// TIA Portal V16 export
// export: Created 2021-11-12T13:31:14.9481279Z, ExportSetting WithDefaults, DisplayName Totally Integrated Automation Portal, DisplayVersion V16 Update 3, DisplayName TIA Portal Version Control Interface, DisplayVersion V16 Update 2, DisplayName TIA Portal Openness, DisplayVersion V16 Update 3, DisplayName SINAMICS Startdrive Advanced, DisplayVersion V16 Update 5, DisplayName SINAMICS Startdrive G130, G150, S120, S150, SINAMICS MV, S210, DisplayVersion V16 Update 5, DisplayName SINAMICS Startdrive G110M, G120, G120C, G120D, G120P, G115D, DisplayVersion V16 Update 5, DisplayName STEP 7 Professional, DisplayVersion V16 Update 3, DisplayName STEP 7 Safety, DisplayVersion V16, DisplayName WinCC UA Professional, DisplayVersion V16 Update 3
FUNCTION_BLOCK "STD_EuchnerDoor"   // FB77, LAD
{ S7_Optimized_Access := 'TRUE' }
VERSION : 0.1
// MICE STD Function Block
// STD_EuchnerDoor MGB2 module
// 
// Version                             Creation date                       Created by
// stored: AutoNumber true, IsIECCheckEnabled false, IsRetainMemResEnabled false, MemoryReserve 100, SetENOAutomatically false, UDAEnableTagReadback false
   VAR_INPUT
      IB_SubModule : "136687_UDT_MSM_Basic.Input";
      IB_LockModule : "UDT_MGB2-L/I_Extended.Input";
      IS_ZoneM : "UDT_Status_main";
      IS_ZoneS : "UDT_Zone_Status_specific";
      IB1LampTest : Bool;   // Lamp test button
      IB1Blinking_1Hz : Bool;   // Tact 1Hz
      IB1Blinking_2Hz : Bool;   // Tact 2Hz
      IB1AckReq : Bool;   // Alarms are resettable
      IB1UlckEn : Bool;   // Unlock enable
      IB1LckEn : Bool;   // Lock enable
      IB1LckMode : Bool;   // Lock mode - 1 can be lock before door is closed
      IB1Start : Bool;   // Start after zone was paused
      IB1AckRequestFromSafety : Bool;   // Safety block SFDoor needs ack
   END_VAR
   VAR_OUTPUT
      OS_Status : Struct
         Main : "UDT_Status_main";
         Specific : "UDT_Door_MGB2_L1_Status_specific";
         Error : "UDT_Error01";
      END_STRUCT;
      OB_SubModule : "136687_UDT_MSM.Output";
      OB_LockModule : "UDT_MGB-L/I.Output";
      OB1AckForSafety : Bool;   // Signal to Safety program
   END_VAR
   VAR
      SS_Alarm : Struct   // Device alarms
         SubModuleS1 : Bool;   // Sub module: Error S1
         LockModuleSM0 : Bool;   // Locking module: Error Sub module 0
         LockModuleSM1 : Bool;   // Locking module: Error Sub module 1
         LockModuleER : Bool;   // Locking module: Error escape release
         LockModuleG : Bool;   // Locking module: Error generally
         Res_0_5 : Bool;
         Res_0_6 : Bool;
         Res_0_7 : Bool;
         Res_1_0 : Bool;
         Res_1_1 : Bool;
         Res_1_2 : Bool;
         Res_1_3 : Bool;
         Res_1_4 : Bool;
         Res_1_5 : Bool;
         Res_1_6 : Bool;
         Res_1_7 : Bool;
      END_STRUCT;
      SS_Warning : Struct   // Device warnings
         Res_0_1 : Bool;
         Res_0_2 : Bool;
         Res_0_3 : Bool;
         Res_0_4 : Bool;
         Res_0_5 : Bool;
         Res_0_6 : Bool;
         Res_0_7 : Bool;
         Res_1_0 : Bool;
         Res_1_1 : Bool;
         Res_1_2 : Bool;
         Res_1_3 : Bool;
         Res_1_4 : Bool;
         Res_1_5 : Bool;
         Res_1_6 : Bool;
         Res_1_7 : Bool;
      END_STRUCT;
      SS_Edge : Array[0..9] of Bool;
      ST_PauseTON { S7_SetPoint := 'True'} : TON_TIME;   // Timer for pause
      ST_ACkSafetyTP : TP_TIME;   // Ack locked doors
      SB1CollError : Bool;   // Collective error from device
      SB1EStopLamp : Bool;   // E-Stop lamp
      SB0Lock : Bool;   // Lock signal (output)
      SB1RequestLock : Bool;   // Request to lock
      SB1RequestUnlock : Bool;   // Request to unlock
      SB1ResetLamp : Bool;   // Lock and reset alarm lamp
      SB1RequestLamp : Bool;   // Request to open lamp
      SB1RequestPause : Bool;   // Request to pause
      SB1ReadyToLock : Bool;
      SB1ReadyToOpen : Bool;
   END_VAR
   VAR_TEMP
      TS_Status : Struct
         Main : "UDT_Status_main";
         Specific : "UDT_Door_MGB2_L1_Status_specific";
         Error : "UDT_Error01";
      END_STRUCT;
   END_VAR
   VAR_TEMP   // added for the SCL form of the ladder/FBD networks
      _w1 : Bool;
   END_VAR
BEGIN

REGION Network 1: Clear temporary TS_Status - Main, Specific
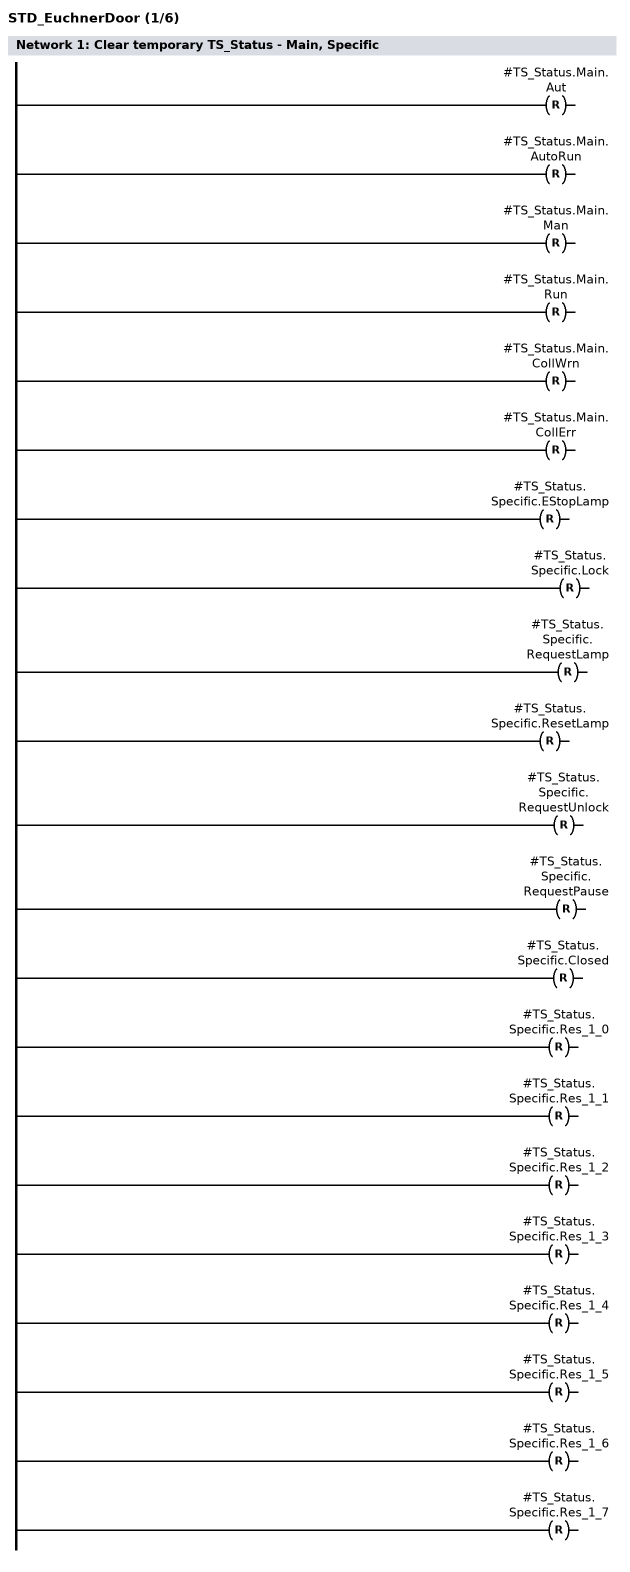
   RUNG wire#powerrail
      R_Coil( #TS_Status.Main.Aut )
   END_RUNG
   RUNG wire#powerrail
      R_Coil( #TS_Status.Main.AutoRun )
   END_RUNG
   RUNG wire#powerrail
      R_Coil( #TS_Status.Main.Man )
   END_RUNG
   RUNG wire#powerrail
      R_Coil( #TS_Status.Main.Run )
   END_RUNG
   RUNG wire#powerrail
      R_Coil( #TS_Status.Main.CollWrn )
   END_RUNG
   RUNG wire#powerrail
      R_Coil( #TS_Status.Main.CollErr )
   END_RUNG
   RUNG wire#powerrail
      R_Coil( #TS_Status.Specific.EStopLamp )
   END_RUNG
   RUNG wire#powerrail
      R_Coil( #TS_Status.Specific.Lock )
   END_RUNG
   RUNG wire#powerrail
      R_Coil( #TS_Status.Specific.RequestLamp )
   END_RUNG
   RUNG wire#powerrail
      R_Coil( #TS_Status.Specific.ResetLamp )
   END_RUNG
   RUNG wire#powerrail
      R_Coil( #TS_Status.Specific.RequestUnlock )
   END_RUNG
   RUNG wire#powerrail
      R_Coil( #TS_Status.Specific.RequestPause )
   END_RUNG
   RUNG wire#powerrail
      R_Coil( #TS_Status.Specific.Closed )
   END_RUNG
   RUNG wire#powerrail
      R_Coil( #TS_Status.Specific.Res_1_0 )
   END_RUNG
   RUNG wire#powerrail
      R_Coil( #TS_Status.Specific.Res_1_1 )
   END_RUNG
   RUNG wire#powerrail
      R_Coil( #TS_Status.Specific.Res_1_2 )
   END_RUNG
   RUNG wire#powerrail
      R_Coil( #TS_Status.Specific.Res_1_3 )
   END_RUNG
   RUNG wire#powerrail
      R_Coil( #TS_Status.Specific.Res_1_4 )
   END_RUNG
   RUNG wire#powerrail
      R_Coil( #TS_Status.Specific.Res_1_5 )
   END_RUNG
   RUNG wire#powerrail
      R_Coil( #TS_Status.Specific.Res_1_6 )
   END_RUNG
   RUNG wire#powerrail
      R_Coil( #TS_Status.Specific.Res_1_7 )
   END_RUNG
   // the same network as SCL:
   #TS_Status.Main.Aut := FALSE;
   #TS_Status.Main.AutoRun := FALSE;
   #TS_Status.Main.Man := FALSE;
   #TS_Status.Main.Run := FALSE;
   #TS_Status.Main.CollWrn := FALSE;
   #TS_Status.Main.CollErr := FALSE;
   #TS_Status.Specific.EStopLamp := FALSE;
   #TS_Status.Specific.Lock := FALSE;
   #TS_Status.Specific.RequestLamp := FALSE;
   #TS_Status.Specific.ResetLamp := FALSE;
   #TS_Status.Specific.RequestUnlock := FALSE;
   #TS_Status.Specific.RequestPause := FALSE;
   #TS_Status.Specific.Closed := FALSE;
   #TS_Status.Specific.Res_1_0 := FALSE;
   #TS_Status.Specific.Res_1_1 := FALSE;
   #TS_Status.Specific.Res_1_2 := FALSE;
   #TS_Status.Specific.Res_1_3 := FALSE;
   #TS_Status.Specific.Res_1_4 := FALSE;
   #TS_Status.Specific.Res_1_5 := FALSE;
   #TS_Status.Specific.Res_1_6 := FALSE;
   #TS_Status.Specific.Res_1_7 := FALSE;
END_REGION

REGION Network 2: Collective error of device
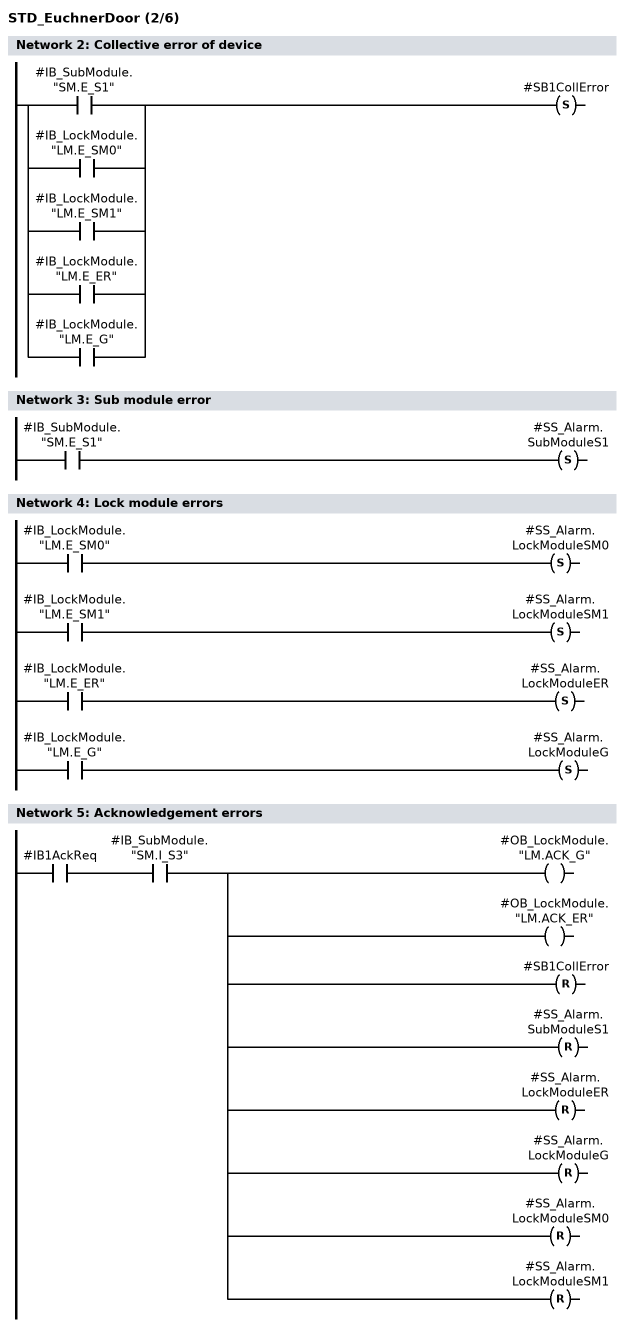
   RUNG wire#powerrail
      Contact( #IB_SubModule."SM.E_S1" )
      wire#w1
      S_Coil( #SB1CollError )
   END_RUNG
   RUNG wire#powerrail
      Contact( #IB_LockModule."LM.E_SM0" )
   END_RUNG wire#w1
   RUNG wire#powerrail
      Contact( #IB_LockModule."LM.E_SM1" )
   END_RUNG wire#w1
   RUNG wire#powerrail
      Contact( #IB_LockModule."LM.E_ER" )
   END_RUNG wire#w1
   RUNG wire#powerrail
      Contact( #IB_LockModule."LM.E_G" )
   END_RUNG wire#w1
   // the same network as SCL:
   IF #IB_SubModule."SM.E_S1" OR #IB_LockModule."LM.E_SM0" OR #IB_LockModule."LM.E_SM1" OR #IB_LockModule."LM.E_ER" OR #IB_LockModule."LM.E_G" THEN
       #SB1CollError := TRUE;
   END_IF;
END_REGION

REGION Network 3: Sub module error
   RUNG wire#powerrail
      Contact( #IB_SubModule."SM.E_S1" )
      S_Coil( #SS_Alarm.SubModuleS1 )
   END_RUNG
   // the same network as SCL:
   IF #IB_SubModule."SM.E_S1" THEN #SS_Alarm.SubModuleS1 := TRUE; END_IF;
END_REGION

REGION Network 4: Lock module errors
   RUNG wire#powerrail
      Contact( #IB_LockModule."LM.E_SM0" )
      S_Coil( #SS_Alarm.LockModuleSM0 )
   END_RUNG
   RUNG wire#powerrail
      Contact( #IB_LockModule."LM.E_SM1" )
      S_Coil( #SS_Alarm.LockModuleSM1 )
   END_RUNG
   RUNG wire#powerrail
      Contact( #IB_LockModule."LM.E_ER" )
      S_Coil( #SS_Alarm.LockModuleER )
   END_RUNG
   RUNG wire#powerrail
      Contact( #IB_LockModule."LM.E_G" )
      S_Coil( #SS_Alarm.LockModuleG )
   END_RUNG
   // the same network as SCL:
   IF #IB_LockModule."LM.E_SM0" THEN #SS_Alarm.LockModuleSM0 := TRUE; END_IF;
   IF #IB_LockModule."LM.E_SM1" THEN #SS_Alarm.LockModuleSM1 := TRUE; END_IF;
   IF #IB_LockModule."LM.E_ER" THEN #SS_Alarm.LockModuleER := TRUE; END_IF;
   IF #IB_LockModule."LM.E_G" THEN #SS_Alarm.LockModuleG := TRUE; END_IF;
END_REGION

REGION Network 5: Acknowledgement errors
   RUNG wire#powerrail
      Contact( #IB1AckReq )
      Contact( #IB_SubModule."SM.I_S3" )
      wire#w1
      Coil( #OB_LockModule."LM.ACK_G" )
   END_RUNG
   RUNG wire#w1
      Coil( #OB_LockModule."LM.ACK_ER" )
   END_RUNG
   RUNG wire#w1
      R_Coil( #SB1CollError )
   END_RUNG
   RUNG wire#w1
      R_Coil( #SS_Alarm.SubModuleS1 )
   END_RUNG
   RUNG wire#w1
      R_Coil( #SS_Alarm.LockModuleER )
   END_RUNG
   RUNG wire#w1
      R_Coil( #SS_Alarm.LockModuleG )
   END_RUNG
   RUNG wire#w1
      R_Coil( #SS_Alarm.LockModuleSM0 )
   END_RUNG
   RUNG wire#w1
      R_Coil( #SS_Alarm.LockModuleSM1 )
   END_RUNG
   // the same network as SCL:
   #OB_LockModule."LM.ACK_G" := #IB1AckReq AND #IB_SubModule."SM.I_S3";
   #OB_LockModule."LM.ACK_ER" := #OB_LockModule."LM.ACK_G";
   IF #OB_LockModule."LM.ACK_G" THEN
       #SB1CollError := FALSE;
       #SS_Alarm.SubModuleS1 := FALSE;
       #SS_Alarm.LockModuleER := FALSE;
       #SS_Alarm.LockModuleG := FALSE;
       #SS_Alarm.LockModuleSM0 := FALSE;
       #SS_Alarm.LockModuleSM1 := FALSE;
   END_IF;
END_REGION

REGION Network 6: Red lamp - E-Stop
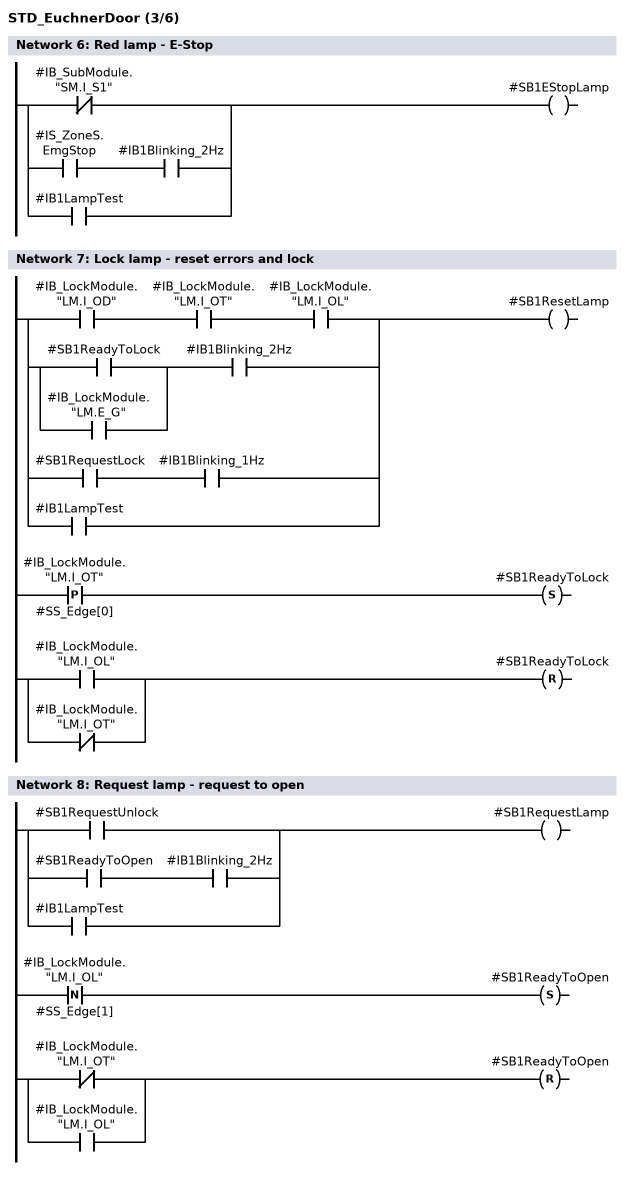
   RUNG wire#powerrail
      I_Contact( #IB_SubModule."SM.I_S1" )
      wire#w1
      Coil( #SB1EStopLamp )
   END_RUNG
   RUNG wire#powerrail
      Contact( #IS_ZoneS.EmgStop )
      Contact( #IB1Blinking_2Hz )
   END_RUNG wire#w1
   RUNG wire#powerrail
      Contact( #IB1LampTest )
   END_RUNG wire#w1
   // the same network as SCL:
   #SB1EStopLamp := NOT #IB_SubModule."SM.I_S1" OR (#IS_ZoneS.EmgStop AND #IB1Blinking_2Hz) OR #IB1LampTest;
END_REGION

REGION Network 7: Lock lamp - reset errors and lock
   RUNG wire#powerrail
      Contact( #IB_LockModule."LM.I_OD" )
      Contact( #IB_LockModule."LM.I_OT" )
      Contact( #IB_LockModule."LM.I_OL" )
      wire#w1
      Coil( #SB1ResetLamp )
   END_RUNG
   RUNG wire#powerrail
      Contact( #SB1ReadyToLock )
      wire#w2
      Contact( #IB1Blinking_2Hz )
   END_RUNG wire#w1
   RUNG wire#powerrail
      Contact( #IB_LockModule."LM.E_G" )
   END_RUNG wire#w2
   RUNG wire#powerrail
      Contact( #SB1RequestLock )
      Contact( #IB1Blinking_1Hz )
   END_RUNG wire#w1
   RUNG wire#powerrail
      Contact( #IB1LampTest )
   END_RUNG wire#w1
   RUNG wire#powerrail
      P_Contact(operand := #IB_LockModule."LM.I_OT", bit := #SS_Edge[0])
      S_Coil( #SB1ReadyToLock )
   END_RUNG
   RUNG wire#powerrail
      Contact( #IB_LockModule."LM.I_OL" )
      wire#w3
      R_Coil( #SB1ReadyToLock )
   END_RUNG
   RUNG wire#powerrail
      I_Contact( #IB_LockModule."LM.I_OT" )
   END_RUNG wire#w3
   // the same network as SCL:
   #SB1ResetLamp := (#IB_LockModule."LM.I_OD" AND #IB_LockModule."LM.I_OT" AND #IB_LockModule."LM.I_OL") OR ((#SB1ReadyToLock OR #IB_LockModule."LM.E_G") AND #IB1Blinking_2Hz) OR (#SB1RequestLock AND #IB1Blinking_1Hz) OR #IB1LampTest;
   #_w1 := #IB_LockModule."LM.I_OT" AND NOT #SS_Edge[0];   // rising edge of #IB_LockModule."LM.I_OT"
   #SS_Edge[0] := #IB_LockModule."LM.I_OT";
   IF #_w1 THEN #SB1ReadyToLock := TRUE; END_IF;
   IF #IB_LockModule."LM.I_OL" OR NOT #IB_LockModule."LM.I_OT" THEN #SB1ReadyToLock := FALSE; END_IF;
END_REGION

REGION Network 8: Request lamp - request to open
   RUNG wire#powerrail
      Contact( #SB1RequestUnlock )
      wire#w1
      Coil( #SB1RequestLamp )
   END_RUNG
   RUNG wire#powerrail
      Contact( #SB1ReadyToOpen )
      Contact( #IB1Blinking_2Hz )
   END_RUNG wire#w1
   RUNG wire#powerrail
      Contact( #IB1LampTest )
   END_RUNG wire#w1
   RUNG wire#powerrail
      N_Contact(operand := #IB_LockModule."LM.I_OL", bit := #SS_Edge[1])
      S_Coil( #SB1ReadyToOpen )
   END_RUNG
   RUNG wire#powerrail
      I_Contact( #IB_LockModule."LM.I_OT" )
      wire#w2
      R_Coil( #SB1ReadyToOpen )
   END_RUNG
   RUNG wire#powerrail
      Contact( #IB_LockModule."LM.I_OL" )
   END_RUNG wire#w2
   // the same network as SCL:
   #SB1RequestLamp := #SB1RequestUnlock OR (#SB1ReadyToOpen AND #IB1Blinking_2Hz) OR #IB1LampTest;
   #_w1 := NOT #IB_LockModule."LM.I_OL" AND #SS_Edge[1];   // falling edge of #IB_LockModule."LM.I_OL"
   #SS_Edge[1] := #IB_LockModule."LM.I_OL";
   IF #_w1 THEN #SB1ReadyToOpen := TRUE; END_IF;
   IF NOT #IB_LockModule."LM.I_OT" OR #IB_LockModule."LM.I_OL" THEN #SB1ReadyToOpen := FALSE; END_IF;
END_REGION

REGION Network 9: Request to lock
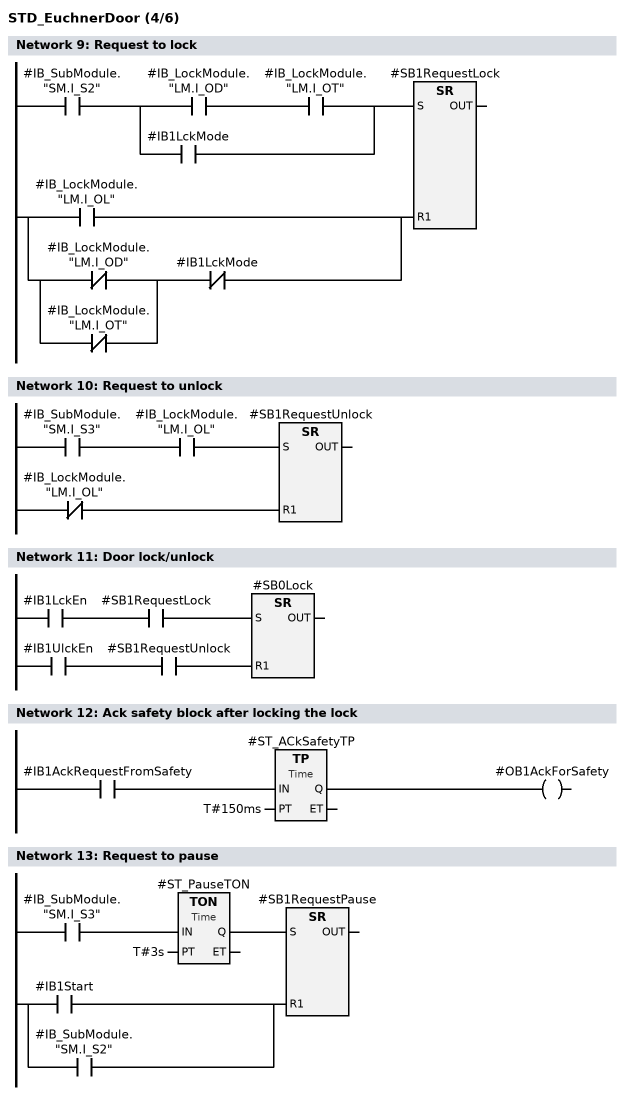
   RUNG wire#powerrail
      Contact( #IB_SubModule."SM.I_S2" )
      wire#w1
      Contact( #IB_LockModule."LM.I_OD" )
      Contact( #IB_LockModule."LM.I_OT" )
      wire#w2
      S_SR(operand := #SB1RequestLock, r1 := wire#w4)
   END_RUNG
   RUNG wire#w1
      Contact( #IB1LckMode )
   END_RUNG wire#w2
   RUNG wire#powerrail
      Contact( #IB_LockModule."LM.I_OL" )
   END_RUNG wire#w4
   RUNG wire#powerrail
      I_Contact( #IB_LockModule."LM.I_OD" )
      wire#w3
      I_Contact( #IB1LckMode )
   END_RUNG wire#w4
   RUNG wire#powerrail
      I_Contact( #IB_LockModule."LM.I_OT" )
   END_RUNG wire#w3
   // the same network as SCL:
   IF #IB_SubModule."SM.I_S2" AND ((#IB_LockModule."LM.I_OD" AND #IB_LockModule."LM.I_OT") OR #IB1LckMode) THEN
       #SB1RequestLock := TRUE;   // SR flip-flop
   END_IF;
   IF #IB_LockModule."LM.I_OL" OR ((NOT #IB_LockModule."LM.I_OD" OR NOT #IB_LockModule."LM.I_OT") AND NOT #IB1LckMode) THEN
       #SB1RequestLock := FALSE;
   END_IF;
END_REGION

REGION Network 10: Request to unlock
   RUNG wire#powerrail
      Contact( #IB_SubModule."SM.I_S3" )
      Contact( #IB_LockModule."LM.I_OL" )
      S_SR(operand := #SB1RequestUnlock, r1 := wire#w1)
   END_RUNG
   RUNG wire#powerrail
      I_Contact( #IB_LockModule."LM.I_OL" )
   END_RUNG wire#w1
   // the same network as SCL:
   IF #IB_SubModule."SM.I_S3" AND #IB_LockModule."LM.I_OL" THEN
       #SB1RequestUnlock := TRUE;   // SR flip-flop
   END_IF;
   IF NOT #IB_LockModule."LM.I_OL" THEN #SB1RequestUnlock := FALSE; END_IF;
END_REGION

REGION Network 11: Door lock/unlock
   RUNG wire#powerrail
      Contact( #IB1LckEn )
      Contact( #SB1RequestLock )
      S_SR(operand := #SB0Lock, r1 := wire#w1)
   END_RUNG
   RUNG wire#powerrail
      Contact( #IB1UlckEn )
      Contact( #SB1RequestUnlock )
   END_RUNG wire#w1
   // the same network as SCL:
   IF #IB1LckEn AND #SB1RequestLock THEN
       #SB0Lock := TRUE;   // SR flip-flop
   END_IF;
   IF #IB1UlckEn AND #SB1RequestUnlock THEN #SB0Lock := FALSE; END_IF;
END_REGION

REGION Network 12: Ack safety block after locking the lock
   RUNG wire#powerrail
      Contact( #IB1AckRequestFromSafety )
      { S7_Templates := "time_type := Time" } #ST_ACkSafetyTP.TP(pt := T#150ms, et =>)
      Coil( #OB1AckForSafety )
   END_RUNG
   // the same network as SCL:
   #ST_ACkSafetyTP(IN := #IB1AckRequestFromSafety, PT := T#150ms);   // TP
   #OB1AckForSafety := #ST_ACkSafetyTP.Q;
END_REGION

REGION Network 13: Request to pause
   RUNG wire#powerrail
      Contact( #IB_SubModule."SM.I_S3" )
      { S7_Templates := "time_type := Time" } #ST_PauseTON.TON(pt := T#3s, et =>)
      S_SR(operand := #SB1RequestPause, r1 := wire#w1)
   END_RUNG
   RUNG wire#powerrail
      Contact( #IB1Start )
   END_RUNG wire#w1
   RUNG wire#powerrail
      Contact( #IB_SubModule."SM.I_S2" )
   END_RUNG wire#w1
   // the same network as SCL:
   #ST_PauseTON(IN := #IB_SubModule."SM.I_S3", PT := T#3s);   // TON
   IF #ST_PauseTON.Q THEN
       #SB1RequestPause := TRUE;   // SR flip-flop
   END_IF;
   IF #IB1Start OR #IB_SubModule."SM.I_S2" THEN #SB1RequestPause := FALSE; END_IF;
END_REGION

REGION Network 14: Copy static variables to output variables
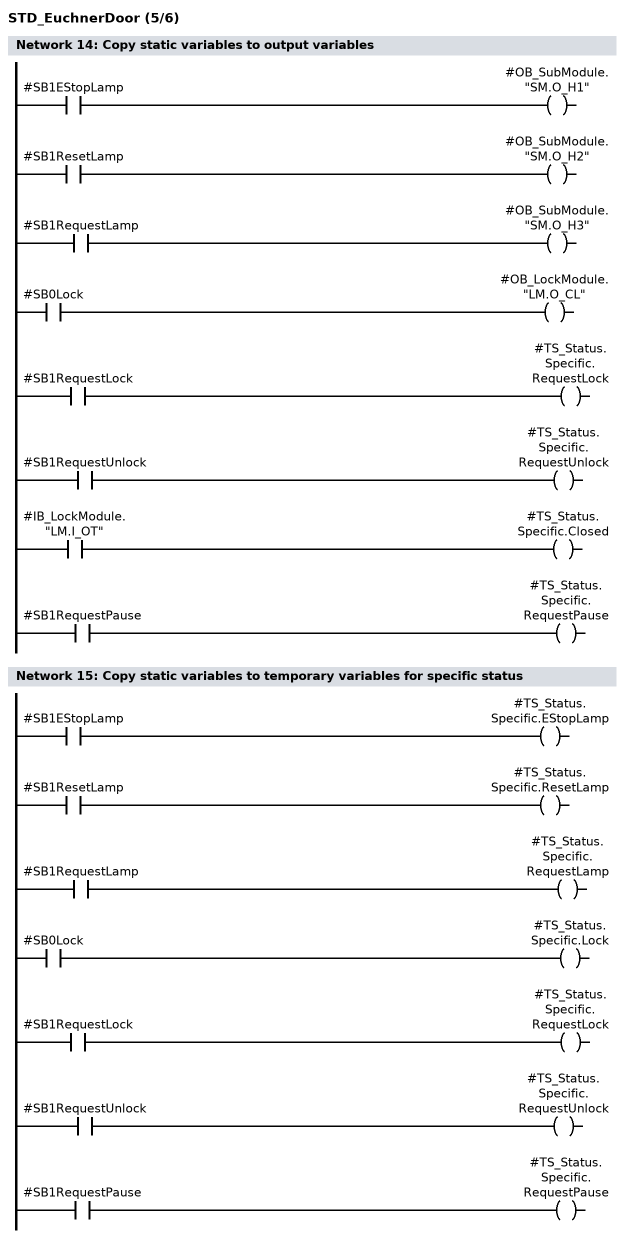
   RUNG wire#powerrail
      Contact( #SB1EStopLamp )
      Coil( #OB_SubModule."SM.O_H1" )
   END_RUNG
   RUNG wire#powerrail
      Contact( #SB1ResetLamp )
      Coil( #OB_SubModule."SM.O_H2" )
   END_RUNG
   RUNG wire#powerrail
      Contact( #SB1RequestLamp )
      Coil( #OB_SubModule."SM.O_H3" )
   END_RUNG
   RUNG wire#powerrail
      Contact( #SB0Lock )
      Coil( #OB_LockModule."LM.O_CL" )
   END_RUNG
   RUNG wire#powerrail
      Contact( #SB1RequestLock )
      Coil( #TS_Status.Specific.RequestLock )
   END_RUNG
   RUNG wire#powerrail
      Contact( #SB1RequestUnlock )
      Coil( #TS_Status.Specific.RequestUnlock )
   END_RUNG
   RUNG wire#powerrail
      Contact( #IB_LockModule."LM.I_OT" )
      Coil( #TS_Status.Specific.Closed )
   END_RUNG
   RUNG wire#powerrail
      Contact( #SB1RequestPause )
      Coil( #TS_Status.Specific.RequestPause )
   END_RUNG
   // the same network as SCL:
   #OB_SubModule."SM.O_H1" := #SB1EStopLamp;
   #OB_SubModule."SM.O_H2" := #SB1ResetLamp;
   #OB_SubModule."SM.O_H3" := #SB1RequestLamp;
   #OB_LockModule."LM.O_CL" := #SB0Lock;
   #TS_Status.Specific.RequestLock := #SB1RequestLock;
   #TS_Status.Specific.RequestUnlock := #SB1RequestUnlock;
   #TS_Status.Specific.Closed := #IB_LockModule."LM.I_OT";
   #TS_Status.Specific.RequestPause := #SB1RequestPause;
END_REGION

REGION Network 15: Copy static variables to temporary variables for specific status
   RUNG wire#powerrail
      Contact( #SB1EStopLamp )
      Coil( #TS_Status.Specific.EStopLamp )
   END_RUNG
   RUNG wire#powerrail
      Contact( #SB1ResetLamp )
      Coil( #TS_Status.Specific.ResetLamp )
   END_RUNG
   RUNG wire#powerrail
      Contact( #SB1RequestLamp )
      Coil( #TS_Status.Specific.RequestLamp )
   END_RUNG
   RUNG wire#powerrail
      Contact( #SB0Lock )
      Coil( #TS_Status.Specific.Lock )
   END_RUNG
   RUNG wire#powerrail
      Contact( #SB1RequestLock )
      Coil( #TS_Status.Specific.RequestLock )
   END_RUNG
   RUNG wire#powerrail
      Contact( #SB1RequestUnlock )
      Coil( #TS_Status.Specific.RequestUnlock )
   END_RUNG
   RUNG wire#powerrail
      Contact( #SB1RequestPause )
      Coil( #TS_Status.Specific.RequestPause )
   END_RUNG
   // the same network as SCL:
   #TS_Status.Specific.EStopLamp := #SB1EStopLamp;
   #TS_Status.Specific.ResetLamp := #SB1ResetLamp;
   #TS_Status.Specific.RequestLamp := #SB1RequestLamp;
   #TS_Status.Specific.Lock := #SB0Lock;
   #TS_Status.Specific.RequestLock := #SB1RequestLock;
   #TS_Status.Specific.RequestUnlock := #SB1RequestUnlock;
   #TS_Status.Specific.RequestPause := #SB1RequestPause;
END_REGION

REGION Network 16: Alarms - copy to output structure
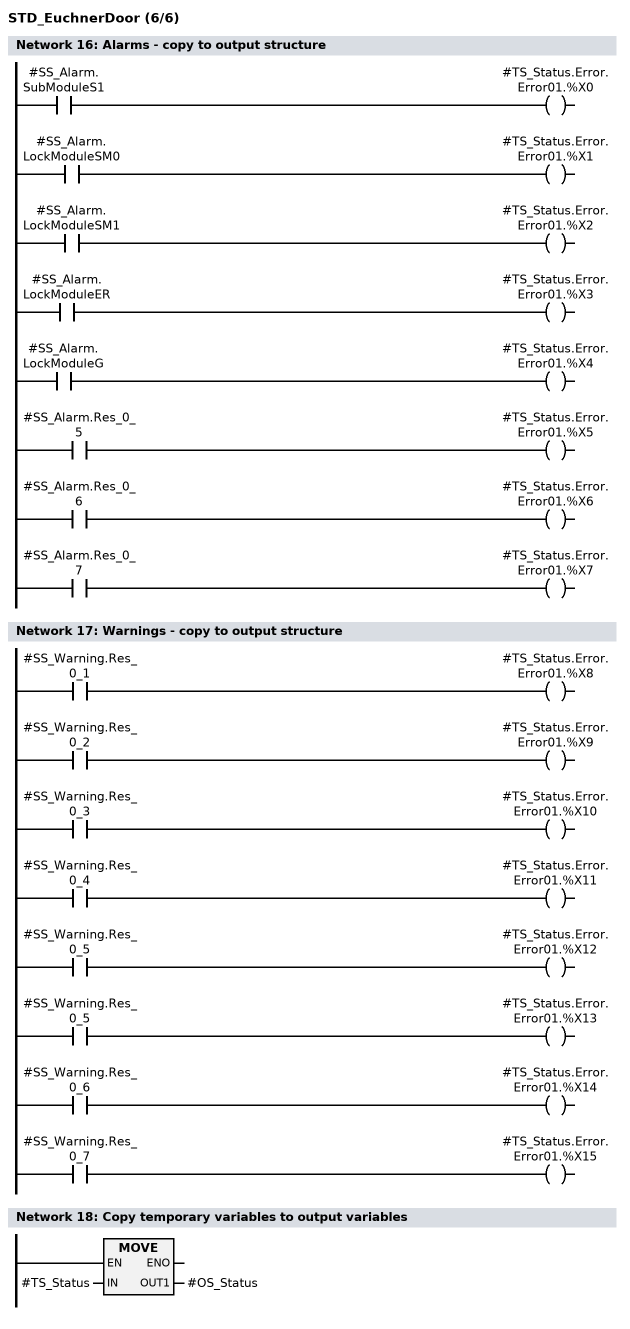
   RUNG wire#powerrail
      Contact( #SS_Alarm.SubModuleS1 )
      Coil( #TS_Status.Error.Error01.%X0 )
   END_RUNG
   RUNG wire#powerrail
      Contact( #SS_Alarm.LockModuleSM0 )
      Coil( #TS_Status.Error.Error01.%X1 )
   END_RUNG
   RUNG wire#powerrail
      Contact( #SS_Alarm.LockModuleSM1 )
      Coil( #TS_Status.Error.Error01.%X2 )
   END_RUNG
   RUNG wire#powerrail
      Contact( #SS_Alarm.LockModuleER )
      Coil( #TS_Status.Error.Error01.%X3 )
   END_RUNG
   RUNG wire#powerrail
      Contact( #SS_Alarm.LockModuleG )
      Coil( #TS_Status.Error.Error01.%X4 )
   END_RUNG
   RUNG wire#powerrail
      Contact( #SS_Alarm.Res_0_5 )
      Coil( #TS_Status.Error.Error01.%X5 )
   END_RUNG
   RUNG wire#powerrail
      Contact( #SS_Alarm.Res_0_6 )
      Coil( #TS_Status.Error.Error01.%X6 )
   END_RUNG
   RUNG wire#powerrail
      Contact( #SS_Alarm.Res_0_7 )
      Coil( #TS_Status.Error.Error01.%X7 )
   END_RUNG
   // the same network as SCL:
   #TS_Status.Error.Error01.%X0 := #SS_Alarm.SubModuleS1;
   #TS_Status.Error.Error01.%X1 := #SS_Alarm.LockModuleSM0;
   #TS_Status.Error.Error01.%X2 := #SS_Alarm.LockModuleSM1;
   #TS_Status.Error.Error01.%X3 := #SS_Alarm.LockModuleER;
   #TS_Status.Error.Error01.%X4 := #SS_Alarm.LockModuleG;
   #TS_Status.Error.Error01.%X5 := #SS_Alarm.Res_0_5;
   #TS_Status.Error.Error01.%X6 := #SS_Alarm.Res_0_6;
   #TS_Status.Error.Error01.%X7 := #SS_Alarm.Res_0_7;
END_REGION

REGION Network 17: Warnings - copy to output structure
   RUNG wire#powerrail
      Contact( #SS_Warning.Res_0_1 )
      Coil( #TS_Status.Error.Error01.%X8 )
   END_RUNG
   RUNG wire#powerrail
      Contact( #SS_Warning.Res_0_2 )
      Coil( #TS_Status.Error.Error01.%X9 )
   END_RUNG
   RUNG wire#powerrail
      Contact( #SS_Warning.Res_0_3 )
      Coil( #TS_Status.Error.Error01.%X10 )
   END_RUNG
   RUNG wire#powerrail
      Contact( #SS_Warning.Res_0_4 )
      Coil( #TS_Status.Error.Error01.%X11 )
   END_RUNG
   RUNG wire#powerrail
      Contact( #SS_Warning.Res_0_5 )
      Coil( #TS_Status.Error.Error01.%X12 )
   END_RUNG
   RUNG wire#powerrail
      Contact( #SS_Warning.Res_0_5 )
      Coil( #TS_Status.Error.Error01.%X13 )
   END_RUNG
   RUNG wire#powerrail
      Contact( #SS_Warning.Res_0_6 )
      Coil( #TS_Status.Error.Error01.%X14 )
   END_RUNG
   RUNG wire#powerrail
      Contact( #SS_Warning.Res_0_7 )
      Coil( #TS_Status.Error.Error01.%X15 )
   END_RUNG
   // the same network as SCL:
   #TS_Status.Error.Error01.%X8 := #SS_Warning.Res_0_1;
   #TS_Status.Error.Error01.%X9 := #SS_Warning.Res_0_2;
   #TS_Status.Error.Error01.%X10 := #SS_Warning.Res_0_3;
   #TS_Status.Error.Error01.%X11 := #SS_Warning.Res_0_4;
   #TS_Status.Error.Error01.%X12 := #SS_Warning.Res_0_5;
   #TS_Status.Error.Error01.%X13 := #SS_Warning.Res_0_5;
   #TS_Status.Error.Error01.%X14 := #SS_Warning.Res_0_6;
   #TS_Status.Error.Error01.%X15 := #SS_Warning.Res_0_7;
END_REGION

REGION Network 18: Copy temporary variables to output variables
   RUNG wire#powerrail
      Move(in := #TS_Status, out1 => #OS_Status)
   END_RUNG
   // the same network as SCL:
   #OS_Status := #TS_Status;
END_REGION
END_FUNCTION_BLOCK
